FUNCTION_BLOCK SIM_ValveWithFB
VAR 
	// Outputs from PLC --> HW
	I_bCmdValveOn AT %I* : BOOL;
	I_bCmdValveOff AT %I* : BOOL;
	
	// Inputs from HW --> PLC
	Q_bStaFeedbackOn AT %Q* : BOOL;
	Q_bStaFeedbackOff AT %Q* : BOOL;
	
	s_tonOn : TON;
	s_tonOff : TON;
	
END_VAR

VAR_OUTPUT
	q_bStaValveOn : BOOL;
	q_bStaValveOff : BOOL;
END_VAR

s_tonOn(IN := I_bCmdValveOn AND NOT(I_bCmdValveOff), PT := T#2S);

IF s_tonOn.Q THEN
	Q_bStaFeedbackOn := TRUE;
ELSIF I_bCmdValveOff THEN
	Q_bStaFeedbackOn := FALSE;
END_IF	
	
s_tonOff(IN := I_bCmdValveOff AND NOT(I_bCmdValveOn), PT := T#2S);

IF s_tonOff.Q THEN
	Q_bStaFeedbackOff := TRUE;
ELSIF I_bCmdValveOn THEN
	Q_bStaFeedbackOff := FALSE;
END_IF

q_bStaValveOn := Q_bStaFeedbackOn;
q_bStaValveOff := Q_bStaFeedbackOff;

END_FUNCTION_BLOCK

(* stored: Version 1.1.0.1, ProductVersion 3.1.4024.12
   POU SIM_ValveWithFB: Id {09601eef-f9e1-47f9-b679-e64bd657cf22}, SpecialFunc None *)
